// TIA Portal V16 export
// export: Created 2023-08-28T09:37:47.7519909Z, ExportSetting WithDefaults, DisplayName Totally Integrated Automation Portal, DisplayVersion V16 Update 6, DisplayName TIA Portal Version Control Interface, DisplayVersion V16 Update 2, DisplayName TIA Portal Openness, DisplayVersion V16 Update 6, DisplayName STEP 7 Professional, DisplayVersion V16 Update 6, DisplayName STEP 7 Safety, DisplayVersion V16, DisplayName WinCC Advanced, DisplayVersion V16 Update 6
DATA_BLOCK "dbWatchDog PLC - WinCC"   // DB61
AUTHOR : rtecmer
VERSION : 0.1
// stored: AutoNumber true, DBAccessibleFromOPCUA true, InstanceOfName 00_S_WatchDog PLC - WinCC, InstanceOfType FB
"00_S_WatchDog PLC - WinCC"
BEGIN
END_DATA_BLOCK
